// Mitsubishi GX Works2 project: MixerDUrcp8pumps   PLC: FX3U/FX3UC

PROGRAM MAIN
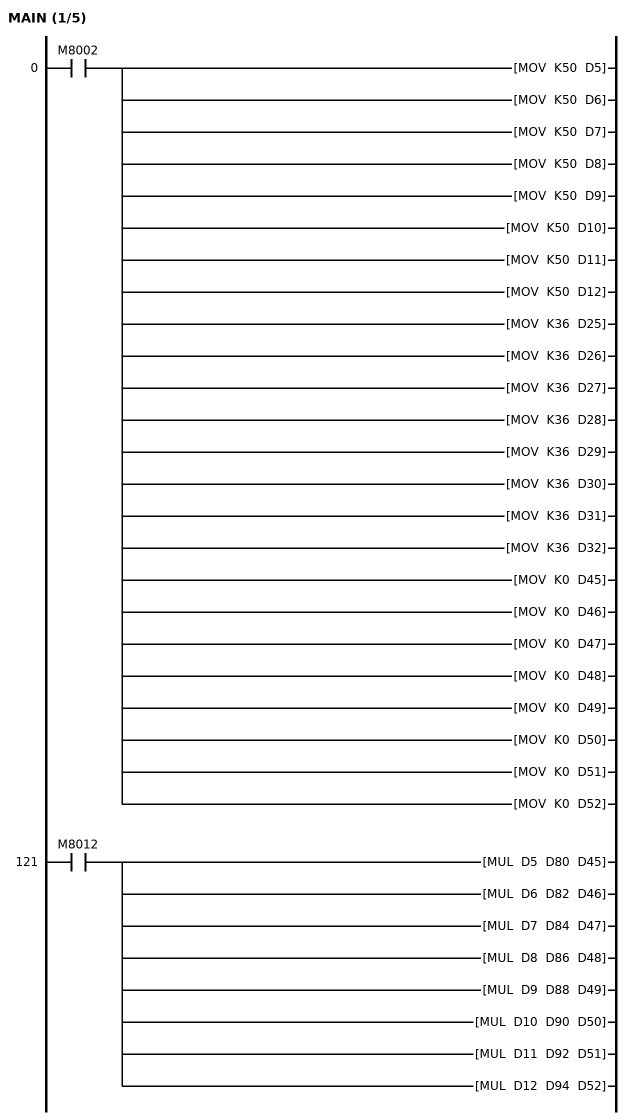
0     LD      M8002
      MOV     K50 D5
      MOV     K50 D6
      MOV     K50 D7
      MOV     K50 D8
      MOV     K50 D9
      MOV     K50 D10
      MOV     K50 D11
      MOV     K50 D12
      MOV     K36 D25
      MOV     K36 D26
      MOV     K36 D27
      MOV     K36 D28
      MOV     K36 D29
      MOV     K36 D30
      MOV     K36 D31
      MOV     K36 D32
      MOV     K0 D45
      MOV     K0 D46
      MOV     K0 D47
      MOV     K0 D48
      MOV     K0 D49
      MOV     K0 D50
      MOV     K0 D51
      MOV     K0 D52
121   LD      M8012
      MUL     D5 D80 D45
      MUL     D6 D82 D46
      MUL     D7 D84 D47
      MUL     D8 D86 D48
      MUL     D9 D88 D49
      MUL     D10 D90 D50
      MUL     D11 D92 D51
      MUL     D12 D94 D52
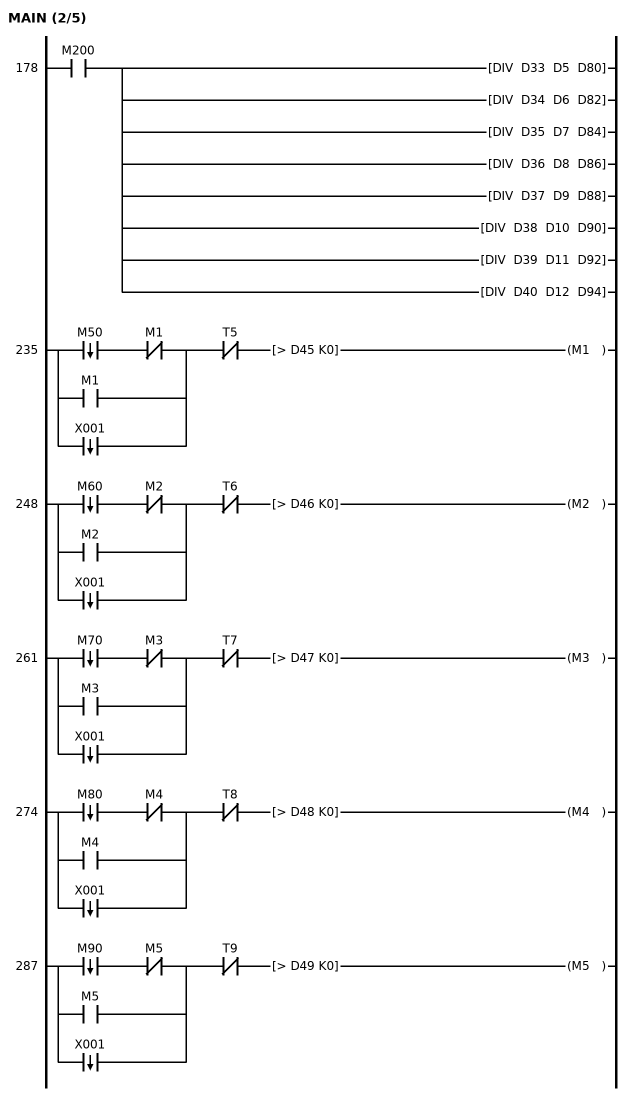
178   LD      M200
      DIV     D33 D5 D80
      DIV     D34 D6 D82
      DIV     D35 D7 D84
      DIV     D36 D8 D86
      DIV     D37 D9 D88
      DIV     D38 D10 D90
      DIV     D39 D11 D92
      DIV     D40 D12 D94
235   LDF     M50
      ANI     M1
      OR      M1
      ORF     X001
      ANI     T5
      AND>    D45 K0
      OUT     M1
248   LDF     M60
      ANI     M2
      OR      M2
      ORF     X001
      ANI     T6
      AND>    D46 K0
      OUT     M2
261   LDF     M70
      ANI     M3
      OR      M3
      ORF     X001
      ANI     T7
      AND>    D47 K0
      OUT     M3
274   LDF     M80
      ANI     M4
      OR      M4
      ORF     X001
      ANI     T8
      AND>    D48 K0
      OUT     M4
287   LDF     M90
      ANI     M5
      OR      M5
      ORF     X001
      ANI     T9
      AND>    D49 K0
      OUT     M5
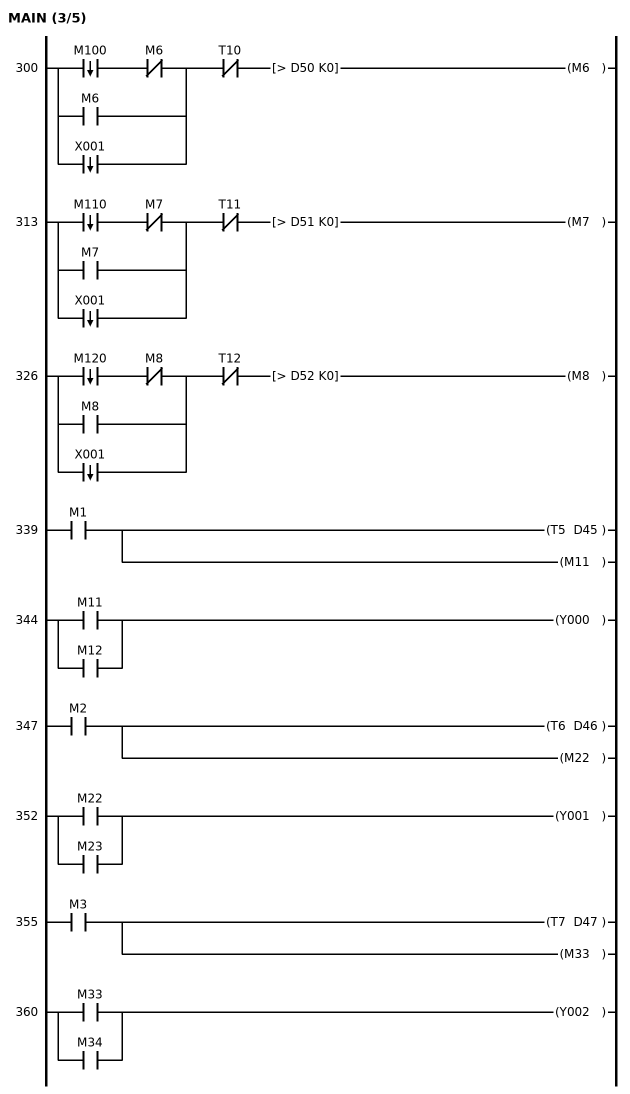
300   LDF     M100
      ANI     M6
      OR      M6
      ORF     X001
      ANI     T10
      AND>    D50 K0
      OUT     M6
313   LDF     M110
      ANI     M7
      OR      M7
      ORF     X001
      ANI     T11
      AND>    D51 K0
      OUT     M7
326   LDF     M120
      ANI     M8
      OR      M8
      ORF     X001
      ANI     T12
      AND>    D52 K0
      OUT     M8
339   LD      M1
      OUT     T5 D45
      OUT     M11
344   LD      M11
      OR      M12
      OUT     Y000
347   LD      M2
      OUT     T6 D46
      OUT     M22
352   LD      M22
      OR      M23
      OUT     Y001
355   LD      M3
      OUT     T7 D47
      OUT     M33
360   LD      M33
      OR      M34
      OUT     Y002
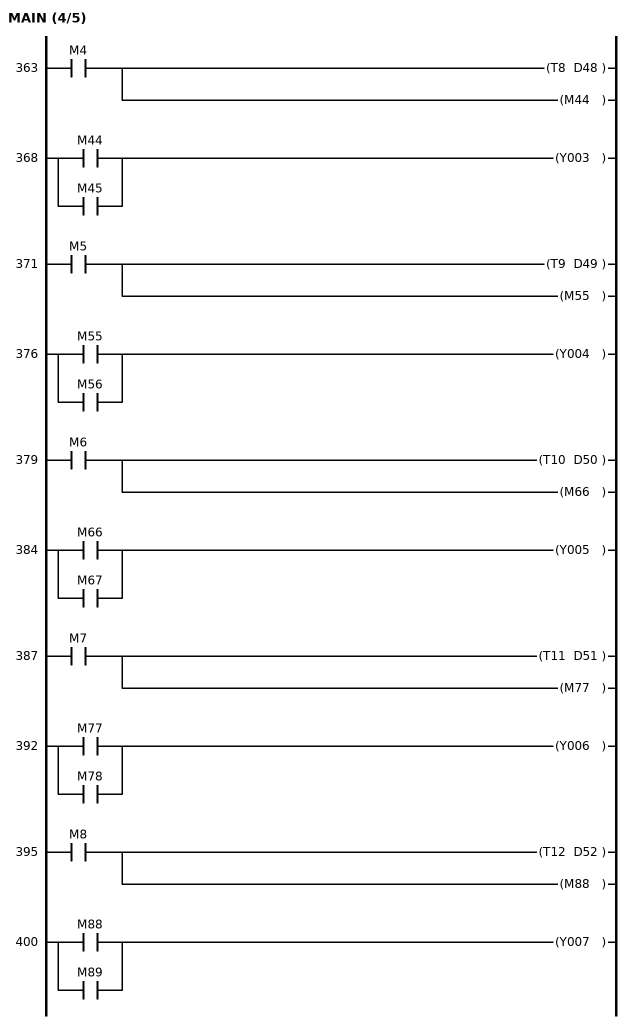
363   LD      M4
      OUT     T8 D48
      OUT     M44
368   LD      M44
      OR      M45
      OUT     Y003
371   LD      M5
      OUT     T9 D49
      OUT     M55
376   LD      M55
      OR      M56
      OUT     Y004
379   LD      M6
      OUT     T10 D50
      OUT     M66
384   LD      M66
      OR      M67
      OUT     Y005
387   LD      M7
      OUT     T11 D51
      OUT     M77
392   LD      M77
      OR      M78
      OUT     Y006
395   LD      M8
      OUT     T12 D52
      OUT     M88
400   LD      M88
      OR      M89
      OUT     Y007
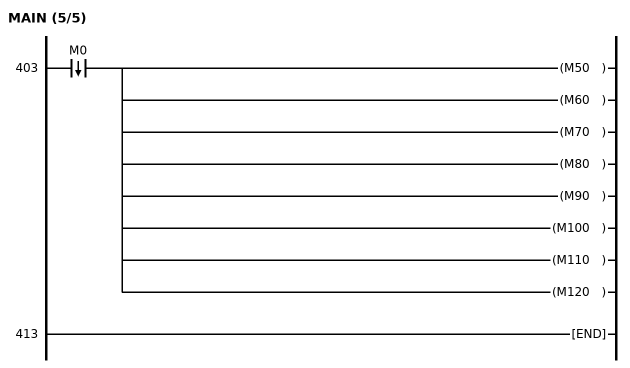
403   LDF     M0
      OUT     M50
      OUT     M60
      OUT     M70
      OUT     M80
      OUT     M90
      OUT     M100
      OUT     M110
      OUT     M120
413   END
END_PROGRAM
